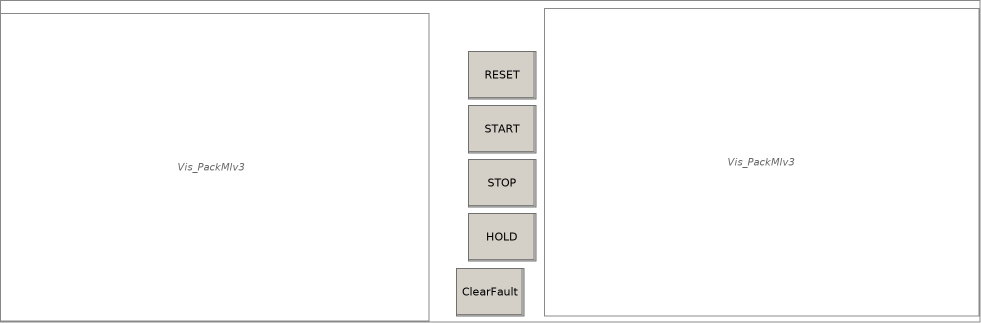
VISUALIZATION Vis_MAIN  // 981x323
    Frame (-6,13 435x308)
        shows Vis_PackMlv3(PML3 := UN01_MachineStateModel)
    Button (468,51 68x48), "RESET"
        tap HMI_Input.Reset
    Button (468,105 68x48), "START"
        tap HMI_Input.Start
    Button (468,159 68x48), "STOP"
        tap HMI_Input.Stop
    Button (468,213 68x48), "HOLD"
        tap HMI_Input.Hold
    Button (456,268 68x48), "ClearFault"
        tap UN01.xDebugReset
    Frame (544,8 435x308)
        shows Vis_PackMlv3(PML3 := UN02_MachineStateModel)
END_VISUALIZATION

(* stored: Version 1.1.0.1, ProductVersion 3.1.4022.16
   Visu Vis_MAIN: Id {44ef75f1-964d-4409-a0e5-e05cb453a9df} *)
